// TIA Portal V17 export
// export: Created 2024-08-29T18:23:44.6087803Z, ExportSetting WithDefaults, DisplayName Totally Integrated Automation Portal, DisplayVersion V17 Update 7, DisplayName TIA Portal Openness, DisplayVersion V17 Update 7, DisplayName TIA Portal Version Control Interface, DisplayVersion V17, DisplayName SINAMICS Startdrive Advanced, DisplayVersion V17 SP2, DisplayName SINAMICS Startdrive G110M, G120, G120C, G120D, G120P, G115D, DisplayVersion V17 SP2, DisplayName SINAMICS Startdrive G130, G150, S120, S150, SINAMICS MV, S210, DisplayVersion V17 SP2, DisplayName STEP 7 Professional, DisplayVersion V17 Update 7, DisplayName STEP 7 Safety, DisplayVersion V17 Update 6, DisplayName WinCC Advanced / Unified PC, DisplayVersion V17 Update 7
FUNCTION "scannerConfiguration" : Void   // FC11, LAD
{ S7_Optimized_Access := 'TRUE' }
VERSION : 0.1
// stored: AutoNumber true, IsIECCheckEnabled false, SetENOAutomatically false, UDAEnableTagReadback false
   VAR_TEMP
      tempScannerOk1 : Bool;
      tempScannerOk2 : Bool;
      tempScannerOk3 : Bool;
   END_VAR
   VAR_TEMP   // added for the SCL form of the ladder/FBD networks
      _w1 : Bool;
      _w2 : Bool;
      _w3 : Bool;
      _w4 : Bool;
      _w5 : Bool;
      _w6 : Bool;
      _w7 : Bool;
      _w8 : Bool;
      _w9 : Bool;
      _w10 : Bool;
      _w11 : Bool;
      _w12 : Bool;
      _w13 : Bool;
      _w14 : Bool;
      _w15 : Bool;
   END_VAR
BEGIN

REGION Network 1: PORT CONFIGURATION
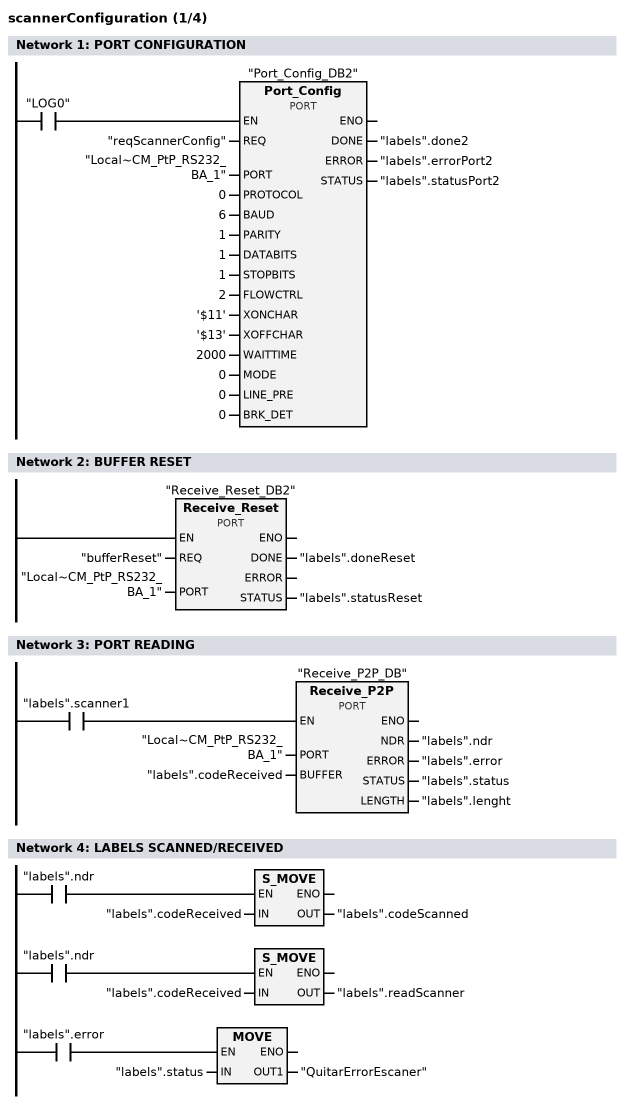
   RUNG wire#powerrail
      Contact( "LOG0" )
      { S7_Templates := "[card := 0, port_type := PORT, word_type := UInt, byte_type := USInt]" } "Port_Config_DB2".Port_Config(REQ := "reqScannerConfig", PORT := "Local~CM_PtP_RS232_BA_1", PROTOCOL := 0, BAUD := 6, PARITY := 1, DATABITS := 1, STOPBITS := 1, FLOWCTRL := 2, XONCHAR := '$11', XOFFCHAR := '$13', WAITTIME := 2000, MODE := 0, LINE_PRE := 0, BRK_DET := 0, DONE => "labels".done2, ERROR => "labels".errorPort2, STATUS => "labels".statusPort2)
   END_RUNG
   // the same network as SCL:
   IF "LOG0" THEN
       "Port_Config_DB2"(REQ := "reqScannerConfig",   // Port_Config
                         PORT := "Local~CM_PtP_RS232_BA_1",
                         PROTOCOL := 0,
                         BAUD := 6,
                         PARITY := 1,
                         DATABITS := 1,
                         STOPBITS := 1,
                         FLOWCTRL := 2,
                         XONCHAR := '$11',
                         XOFFCHAR := '$13',
                         WAITTIME := 2000,
                         MODE := 0,
                         LINE_PRE := 0,
                         BRK_DET := 0,
                         DONE => "labels".done2,
                         ERROR => "labels".errorPort2,
                         STATUS => "labels".statusPort2);
   END_IF;
END_REGION

REGION Network 2: BUFFER RESET
   RUNG wire#powerrail
      { S7_Templates := "[card := 0, port_type := PORT]" } "Receive_Reset_DB2".Receive_Reset(REQ := "bufferReset", PORT := "Local~CM_PtP_RS232_BA_1", DONE => "labels".doneReset, ERROR =>, STATUS => "labels".statusReset)
   END_RUNG
   // the same network as SCL:
   "Receive_Reset_DB2"(REQ := "bufferReset",   // Receive_Reset
                       PORT := "Local~CM_PtP_RS232_BA_1",
                       DONE => "labels".doneReset,
                       STATUS => "labels".statusReset);
END_REGION

REGION Network 3: PORT READING
   RUNG wire#powerrail
      Contact( "labels".scanner1 )
      { S7_Templates := "[card := 0, port_type := PORT, word_type := UInt, any_type := Variant]" } "Receive_P2P_DB".Receive_P2P(PORT := "Local~CM_PtP_RS232_BA_1", BUFFER := "labels".codeReceived, NDR => "labels".ndr, ERROR => "labels".error, STATUS => "labels".status, LENGTH => "labels".lenght)
   END_RUNG
   // the same network as SCL:
   IF "labels".scanner1 THEN
       "Receive_P2P_DB"(PORT := "Local~CM_PtP_RS232_BA_1",   // Receive_P2P
                        BUFFER := "labels".codeReceived,
                        NDR => "labels".ndr,
                        ERROR => "labels".error,
                        STATUS => "labels".status,
                        LENGTH => "labels".lenght);
   END_IF;
END_REGION

REGION Network 4: LABELS SCANNED/RECEIVED
   RUNG wire#powerrail
      Contact( "labels".ndr )
      S_Move(in := "labels".codeReceived, out => "labels".codeScanned)
   END_RUNG
   RUNG wire#powerrail
      Contact( "labels".ndr )
      S_Move(in := "labels".codeReceived, out => "labels".readScanner)
   END_RUNG
   RUNG wire#powerrail
      Contact( "labels".error )
      Move(in := "labels".status, out1 => "QuitarErrorEscaner")
   END_RUNG
   // the same network as SCL:
   IF "labels".ndr THEN
       "labels".codeScanned := "labels".codeReceived;
       "labels".readScanner := "labels".codeReceived;
   END_IF;
   IF "labels".error THEN "QuitarErrorEscaner" := "labels".status; END_IF;
END_REGION

REGION Network 5: SCANNER COMPARISON
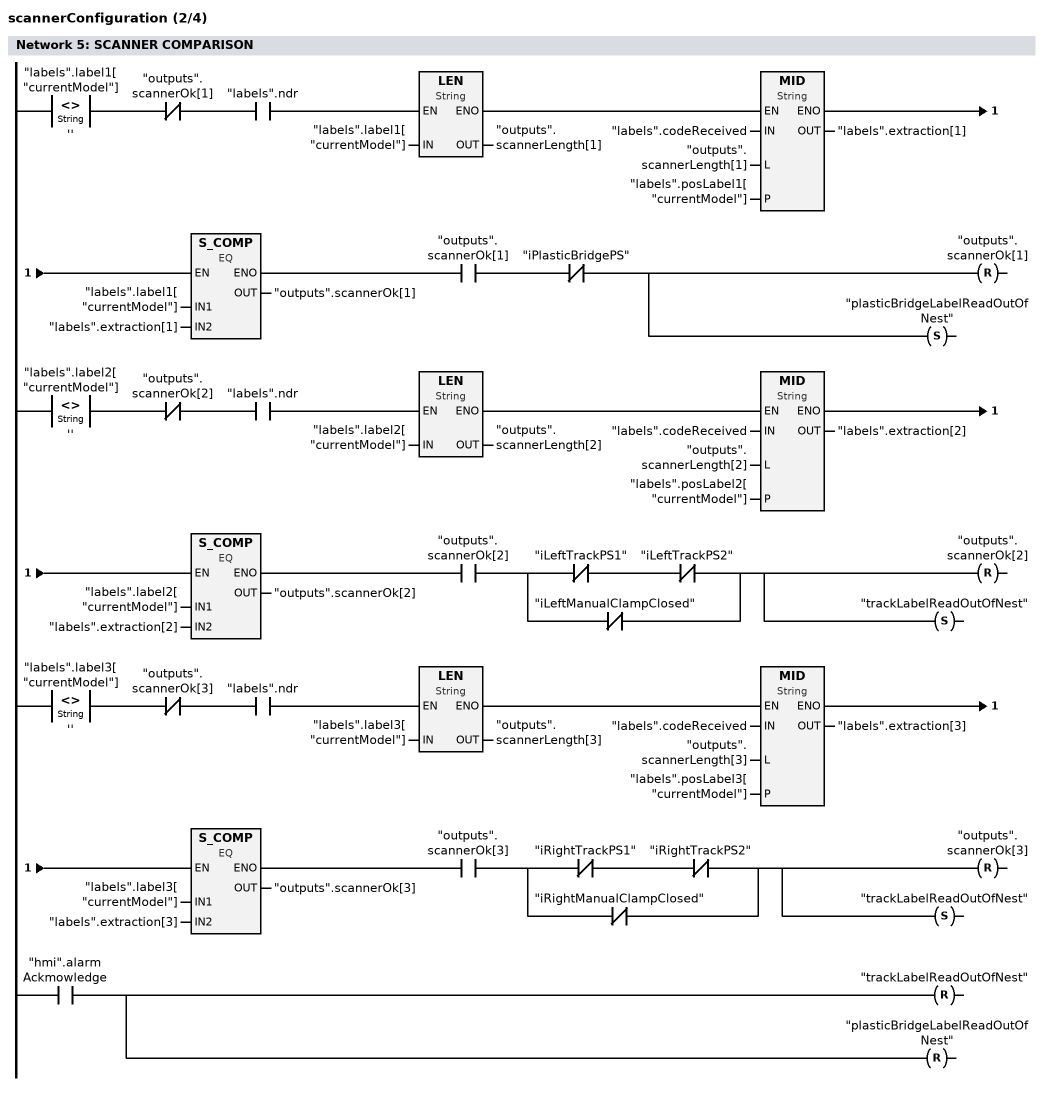
   RUNG wire#powerrail
      { S7_Templates := "SrcType := String" } NE_Contact(in1 := "labels".label1["currentModel"], in2 := '')
      I_Contact( "outputs".scannerOk[1] )
      Contact( "labels".ndr )
      { S7_Templates := "[str_type := String, return_type := Int]" } LEN(IN := "labels".label1["currentModel"], OUT => "outputs".scannerLength[1])
      { S7_Templates := "value_type := String" } MID(IN := "labels".codeReceived, L := "outputs".scannerLength[1], P := "labels".posLabel1["currentModel"], OUT => "labels".extraction[1])
      { S7_Templates := "[relation := EQ, src_type := String]" } S_COMP(IN1 := "labels".label1["currentModel"], IN2 := "labels".extraction[1], OUT => "outputs".scannerOk[1])
      Contact( "outputs".scannerOk[1] )
      I_Contact( "iPlasticBridgePS" )
      wire#w1
      R_Coil( "outputs".scannerOk[1] )
   END_RUNG
   RUNG wire#w1
      S_Coil( "plasticBridgeLabelReadOutOfNest" )
   END_RUNG
   RUNG wire#powerrail
      { S7_Templates := "SrcType := String" } NE_Contact(in1 := "labels".label2["currentModel"], in2 := '')
      I_Contact( "outputs".scannerOk[2] )
      Contact( "labels".ndr )
      { S7_Templates := "[str_type := String, return_type := Int]" } LEN(IN := "labels".label2["currentModel"], OUT => "outputs".scannerLength[2])
      { S7_Templates := "value_type := String" } MID(IN := "labels".codeReceived, L := "outputs".scannerLength[2], P := "labels".posLabel2["currentModel"], OUT => "labels".extraction[2])
      { S7_Templates := "[relation := EQ, src_type := String]" } S_COMP(IN1 := "labels".label2["currentModel"], IN2 := "labels".extraction[2], OUT => "outputs".scannerOk[2])
      Contact( "outputs".scannerOk[2] )
      wire#w2
      I_Contact( "iLeftTrackPS1" )
      I_Contact( "iLeftTrackPS2" )
      wire#w3
      R_Coil( "outputs".scannerOk[2] )
   END_RUNG
   RUNG wire#w2
      I_Contact( "iLeftManualClampClosed" )
   END_RUNG wire#w3
   RUNG wire#w3
      S_Coil( "trackLabelReadOutOfNest" )
   END_RUNG
   RUNG wire#powerrail
      { S7_Templates := "SrcType := String" } NE_Contact(in1 := "labels".label3["currentModel"], in2 := '')
      I_Contact( "outputs".scannerOk[3] )
      Contact( "labels".ndr )
      { S7_Templates := "[str_type := String, return_type := Int]" } LEN(IN := "labels".label3["currentModel"], OUT => "outputs".scannerLength[3])
      { S7_Templates := "value_type := String" } MID(IN := "labels".codeReceived, L := "outputs".scannerLength[3], P := "labels".posLabel3["currentModel"], OUT => "labels".extraction[3])
      { S7_Templates := "[relation := EQ, src_type := String]" } S_COMP(IN1 := "labels".label3["currentModel"], IN2 := "labels".extraction[3], OUT => "outputs".scannerOk[3])
      Contact( "outputs".scannerOk[3] )
      wire#w4
      I_Contact( "iRightTrackPS1" )
      I_Contact( "iRightTrackPS2" )
      wire#w5
      R_Coil( "outputs".scannerOk[3] )
   END_RUNG
   RUNG wire#w4
      I_Contact( "iRightManualClampClosed" )
   END_RUNG wire#w5
   RUNG wire#w5
      S_Coil( "trackLabelReadOutOfNest" )
   END_RUNG
   RUNG wire#powerrail
      Contact( "hmi".alarmAckmowledge )
      wire#w6
      R_Coil( "trackLabelReadOutOfNest" )
   END_RUNG
   RUNG wire#w6
      R_Coil( "plasticBridgeLabelReadOutOfNest" )
   END_RUNG
   // the same network as SCL:
   #_w1 := ("labels".label1["currentModel"] <> '') AND NOT "outputs".scannerOk[1] AND "labels".ndr;
   LEN(EN := #_w1, IN := "labels".label1["currentModel"], OUT => "outputs".scannerLength[1], ENO => #_w2);
   MID(EN := #_w2,
       IN := "labels".codeReceived,
       L := "outputs".scannerLength[1],
       P := "labels".posLabel1["currentModel"],
       OUT => "labels".extraction[1],
       ENO => #_w3);
   S_COMP(EN := #_w3,
          IN1 := "labels".label1["currentModel"],
          IN2 := "labels".extraction[1],
          OUT => "outputs".scannerOk[1],
          ENO => #_w4);
   #_w5 := #_w4 AND "outputs".scannerOk[1] AND NOT "iPlasticBridgePS";
   IF #_w5 THEN
       "outputs".scannerOk[1] := FALSE;
       "plasticBridgeLabelReadOutOfNest" := TRUE;
   END_IF;
   #_w6 := ("labels".label2["currentModel"] <> '') AND NOT "outputs".scannerOk[2] AND "labels".ndr;
   LEN(EN := #_w6, IN := "labels".label2["currentModel"], OUT => "outputs".scannerLength[2], ENO => #_w7);
   MID(EN := #_w7,
       IN := "labels".codeReceived,
       L := "outputs".scannerLength[2],
       P := "labels".posLabel2["currentModel"],
       OUT => "labels".extraction[2],
       ENO => #_w8);
   S_COMP(EN := #_w8,
          IN1 := "labels".label2["currentModel"],
          IN2 := "labels".extraction[2],
          OUT => "outputs".scannerOk[2],
          ENO => #_w9);
   #_w10 := #_w9 AND "outputs".scannerOk[2] AND ((NOT "iLeftTrackPS1" AND NOT "iLeftTrackPS2") OR NOT "iLeftManualClampClosed");
   IF #_w10 THEN
       "outputs".scannerOk[2] := FALSE;
       "trackLabelReadOutOfNest" := TRUE;
   END_IF;
   #_w11 := ("labels".label3["currentModel"] <> '') AND NOT "outputs".scannerOk[3] AND "labels".ndr;
   LEN(EN := #_w11, IN := "labels".label3["currentModel"], OUT => "outputs".scannerLength[3], ENO => #_w12);
   MID(EN := #_w12,
       IN := "labels".codeReceived,
       L := "outputs".scannerLength[3],
       P := "labels".posLabel3["currentModel"],
       OUT => "labels".extraction[3],
       ENO => #_w13);
   S_COMP(EN := #_w13,
          IN1 := "labels".label3["currentModel"],
          IN2 := "labels".extraction[3],
          OUT => "outputs".scannerOk[3],
          ENO => #_w14);
   #_w15 := #_w14 AND "outputs".scannerOk[3] AND ((NOT "iRightTrackPS1" AND NOT "iRightTrackPS2") OR NOT "iRightManualClampClosed");
   IF #_w15 THEN
       "outputs".scannerOk[3] := FALSE;
       "trackLabelReadOutOfNest" := TRUE;
   END_IF;
   IF "hmi".alarmAckmowledge THEN
       "trackLabelReadOutOfNest" := FALSE;
       "plasticBridgeLabelReadOutOfNest" := FALSE;
   END_IF;
END_REGION

REGION Network 6: CHANGE OF STEP SCANNER RESET
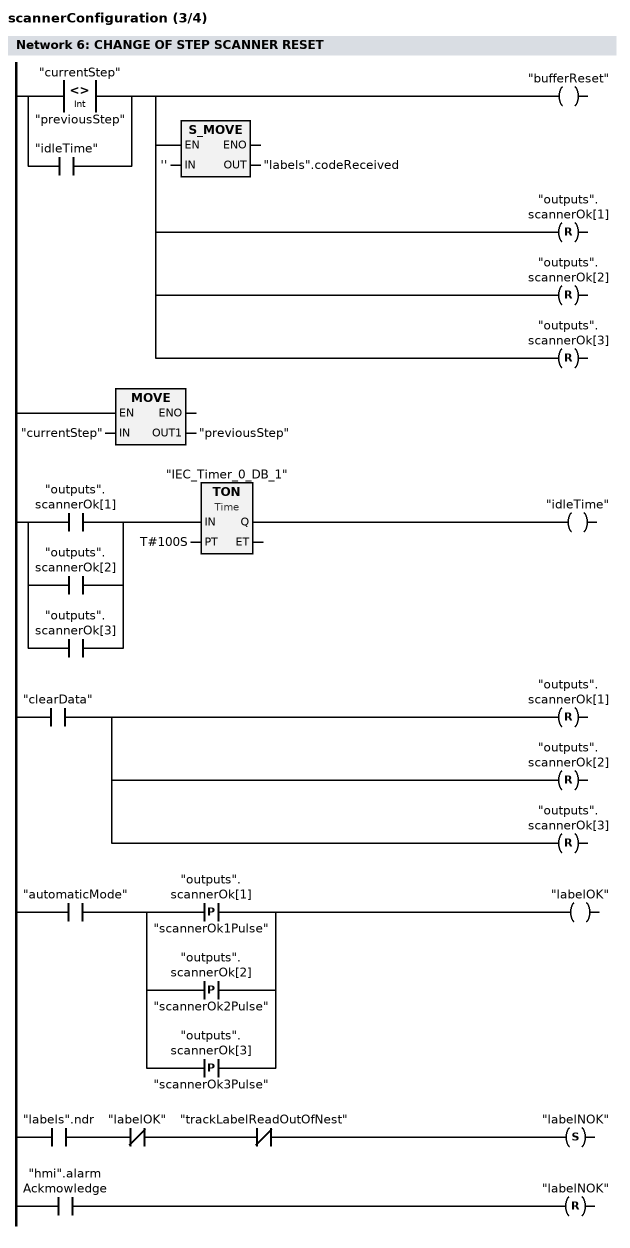
   RUNG wire#powerrail
      { S7_Templates := "SrcType := Int" } NE_Contact(in1 := "currentStep", in2 := "previousStep")
      wire#w1
      Coil( "bufferReset" )
   END_RUNG
   RUNG wire#powerrail
      Contact( "idleTime" )
   END_RUNG wire#w1
   RUNG wire#w1
      S_Move(in := '', out => "labels".codeReceived)
   END_RUNG
   RUNG wire#w1
      R_Coil( "outputs".scannerOk[1] )
   END_RUNG
   RUNG wire#w1
      R_Coil( "outputs".scannerOk[2] )
   END_RUNG
   RUNG wire#w1
      R_Coil( "outputs".scannerOk[3] )
   END_RUNG
   RUNG wire#powerrail
      Move(in := "currentStep", out1 => "previousStep")
   END_RUNG
   RUNG wire#powerrail
      Contact( "outputs".scannerOk[1] )
      wire#w2
      { S7_Templates := "time_type := Time" } "IEC_Timer_0_DB_1".TON(pt := T#100S, et =>)
      Coil( "idleTime" )
   END_RUNG
   RUNG wire#powerrail
      Contact( "outputs".scannerOk[2] )
   END_RUNG wire#w2
   RUNG wire#powerrail
      Contact( "outputs".scannerOk[3] )
   END_RUNG wire#w2
   RUNG wire#powerrail
      Contact( "clearData" )
      wire#w3
      R_Coil( "outputs".scannerOk[1] )
   END_RUNG
   RUNG wire#w3
      R_Coil( "outputs".scannerOk[2] )
   END_RUNG
   RUNG wire#w3
      R_Coil( "outputs".scannerOk[3] )
   END_RUNG
   RUNG wire#powerrail
      Contact( "automaticMode" )
      wire#w4
      P_Contact(operand := "outputs".scannerOk[1], bit := "scannerOk1Pulse")
      wire#w5
      Coil( "labelOK" )
   END_RUNG
   RUNG wire#w4
      P_Contact(operand := "outputs".scannerOk[2], bit := "scannerOk2Pulse")
   END_RUNG wire#w5
   RUNG wire#w4
      P_Contact(operand := "outputs".scannerOk[3], bit := "scannerOk3Pulse")
   END_RUNG wire#w5
   RUNG wire#powerrail
      Contact( "labels".ndr )
      I_Contact( "labelOK" )
      I_Contact( "trackLabelReadOutOfNest" )
      S_Coil( "labelNOK" )
   END_RUNG
   RUNG wire#powerrail
      Contact( "hmi".alarmAckmowledge )
      R_Coil( "labelNOK" )
   END_RUNG
   // the same network as SCL:
   "bufferReset" := ("currentStep" <> "previousStep") OR "idleTime";
   IF "bufferReset" THEN
       "labels".codeReceived := '';
       "outputs".scannerOk[1] := FALSE;
       "outputs".scannerOk[2] := FALSE;
       "outputs".scannerOk[3] := FALSE;
   END_IF;
   "previousStep" := "currentStep";
   "IEC_Timer_0_DB_1".TON(IN := "outputs".scannerOk[1] OR "outputs".scannerOk[2] OR "outputs".scannerOk[3],
                          PT := T#100S);
   "idleTime" := "IEC_Timer_0_DB_1".Q;
   IF "clearData" THEN
       "outputs".scannerOk[1] := FALSE;
       "outputs".scannerOk[2] := FALSE;
       "outputs".scannerOk[3] := FALSE;
   END_IF;
   #_w1 := "automaticMode" AND "outputs".scannerOk[1] AND NOT "scannerOk1Pulse";   // rising edge of "outputs".scannerOk[1]
   "scannerOk1Pulse" := "outputs".scannerOk[1];
   #_w2 := "automaticMode" AND "outputs".scannerOk[2] AND NOT "scannerOk2Pulse";   // rising edge of "outputs".scannerOk[2]
   "scannerOk2Pulse" := "outputs".scannerOk[2];
   #_w3 := "automaticMode" AND "outputs".scannerOk[3] AND NOT "scannerOk3Pulse";   // rising edge of "outputs".scannerOk[3]
   "scannerOk3Pulse" := "outputs".scannerOk[3];
   "labelOK" := #_w1 OR #_w2 OR #_w3;
   IF "labels".ndr AND NOT "labelOK" AND NOT "trackLabelReadOutOfNest" THEN "labelNOK" := TRUE; END_IF;
   IF "hmi".alarmAckmowledge THEN "labelNOK" := FALSE; END_IF;
END_REGION

REGION Network 7: SCANNER DATA LOG
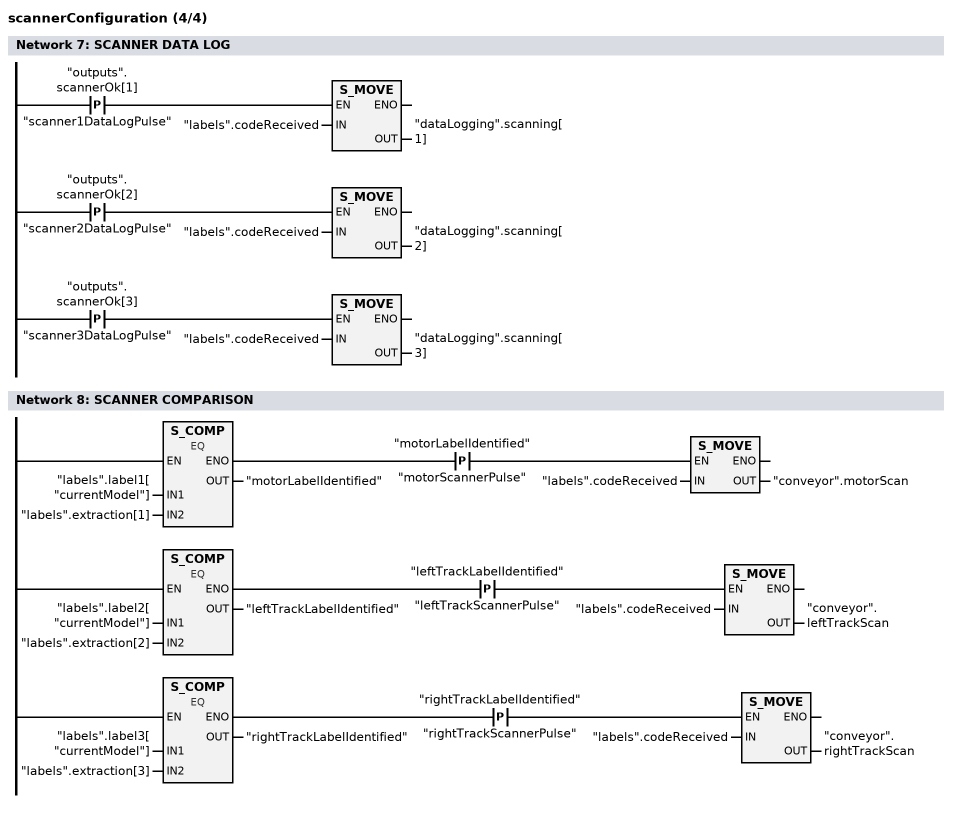
   RUNG wire#powerrail
      P_Contact(operand := "outputs".scannerOk[1], bit := "scanner1DataLogPulse")
      S_Move(in := "labels".codeReceived, out => "dataLogging".scanning[1])
   END_RUNG
   RUNG wire#powerrail
      P_Contact(operand := "outputs".scannerOk[2], bit := "scanner2DataLogPulse")
      S_Move(in := "labels".codeReceived, out => "dataLogging".scanning[2])
   END_RUNG
   RUNG wire#powerrail
      P_Contact(operand := "outputs".scannerOk[3], bit := "scanner3DataLogPulse")
      S_Move(in := "labels".codeReceived, out => "dataLogging".scanning[3])
   END_RUNG
   // the same network as SCL:
   #_w1 := "outputs".scannerOk[1] AND NOT "scanner1DataLogPulse";   // rising edge of "outputs".scannerOk[1]
   "scanner1DataLogPulse" := "outputs".scannerOk[1];
   IF #_w1 THEN "dataLogging".scanning[1] := "labels".codeReceived; END_IF;
   #_w2 := "outputs".scannerOk[2] AND NOT "scanner2DataLogPulse";   // rising edge of "outputs".scannerOk[2]
   "scanner2DataLogPulse" := "outputs".scannerOk[2];
   IF #_w2 THEN "dataLogging".scanning[2] := "labels".codeReceived; END_IF;
   #_w3 := "outputs".scannerOk[3] AND NOT "scanner3DataLogPulse";   // rising edge of "outputs".scannerOk[3]
   "scanner3DataLogPulse" := "outputs".scannerOk[3];
   IF #_w3 THEN "dataLogging".scanning[3] := "labels".codeReceived; END_IF;
END_REGION

REGION Network 8: SCANNER COMPARISON
   RUNG wire#powerrail
      { S7_Templates := "[relation := EQ, src_type := String]" } S_COMP(IN1 := "labels".label1["currentModel"], IN2 := "labels".extraction[1], OUT => "motorLabelIdentified")
      P_Contact(operand := "motorLabelIdentified", bit := "motorScannerPulse")
      S_Move(in := "labels".codeReceived, out => "conveyor".motorScan)
   END_RUNG
   RUNG wire#powerrail
      { S7_Templates := "[relation := EQ, src_type := String]" } S_COMP(IN1 := "labels".label2["currentModel"], IN2 := "labels".extraction[2], OUT => "leftTrackLabelIdentified")
      P_Contact(operand := "leftTrackLabelIdentified", bit := "leftTrackScannerPulse")
      S_Move(in := "labels".codeReceived, out => "conveyor".leftTrackScan)
   END_RUNG
   RUNG wire#powerrail
      { S7_Templates := "[relation := EQ, src_type := String]" } S_COMP(IN1 := "labels".label3["currentModel"], IN2 := "labels".extraction[3], OUT => "rightTrackLabelIdentified")
      P_Contact(operand := "rightTrackLabelIdentified", bit := "rightTrackScannerPulse")
      S_Move(in := "labels".codeReceived, out => "conveyor".rightTrackScan)
   END_RUNG
   // the same network as SCL:
   S_COMP(IN1 := "labels".label1["currentModel"],
          IN2 := "labels".extraction[1],
          OUT => "motorLabelIdentified",
          ENO => #_w1);
   #_w2 := #_w1 AND "motorLabelIdentified" AND NOT "motorScannerPulse";   // rising edge of "motorLabelIdentified"
   "motorScannerPulse" := "motorLabelIdentified";
   IF #_w2 THEN "conveyor".motorScan := "labels".codeReceived; END_IF;
   S_COMP(IN1 := "labels".label2["currentModel"],
          IN2 := "labels".extraction[2],
          OUT => "leftTrackLabelIdentified",
          ENO => #_w3);
   #_w4 := #_w3 AND "leftTrackLabelIdentified" AND NOT "leftTrackScannerPulse";   // rising edge of "leftTrackLabelIdentified"
   "leftTrackScannerPulse" := "leftTrackLabelIdentified";
   IF #_w4 THEN "conveyor".leftTrackScan := "labels".codeReceived; END_IF;
   S_COMP(IN1 := "labels".label3["currentModel"],
          IN2 := "labels".extraction[3],
          OUT => "rightTrackLabelIdentified",
          ENO => #_w5);
   #_w6 := #_w5 AND "rightTrackLabelIdentified" AND NOT "rightTrackScannerPulse";   // rising edge of "rightTrackLabelIdentified"
   "rightTrackScannerPulse" := "rightTrackLabelIdentified";
   IF #_w6 THEN "conveyor".rightTrackScan := "labels".codeReceived; END_IF;
END_REGION
END_FUNCTION
